FUNCTION_BLOCK Separator (* Basic Function Block Type *)
  (* Standard: 61499-2 *)
  (* Version 0.0, 2015-03-24, 4DIAC-IDE, 4DIAC-Consortium *)
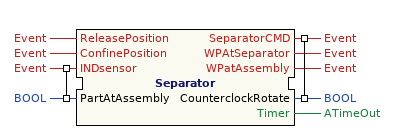
  EVENT_INPUT
    ReleasePosition;
    ConfinePosition;
    INDsensor WITH PartAtAssembly;
  END_EVENT
  EVENT_OUTPUT
    SeparatorCMD WITH CounterclockRotate;
    WPAtSeparator;
    WPatAssembly;
  END_EVENT
  VAR_INPUT
    PartAtAssembly : BOOL;
  END_VAR
  VAR_OUTPUT
    CounterclockRotate : BOOL;
  END_VAR
  PLUGS
    Timer : ATimeOut;
  END_PLUGS
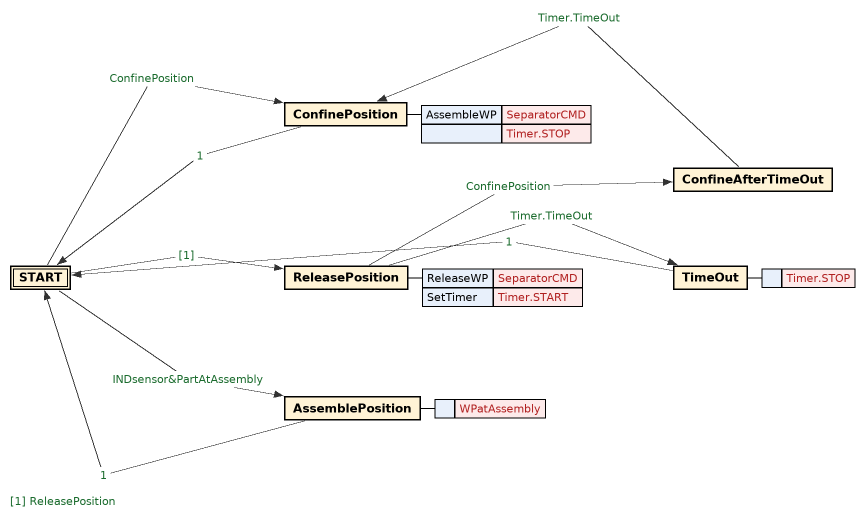
  EC_STATES
    START; (* Initial State *)
    ReleasePosition : ReleaseWP -> SeparatorCMD, SetTimer -> Timer.START;
    AssemblePosition : -> WPatAssembly;
    ConfinePosition : AssembleWP -> SeparatorCMD, -> Timer.STOP;
    TimeOut : -> Timer.STOP;
    ConfineAfterTimeOut;
  END_STATES
  EC_TRANSITIONS
    START TO ReleasePosition := ReleasePosition;
    ConfinePosition TO START := 1;
    AssemblePosition TO START := 1;
    TimeOut TO START := 1;
    ReleasePosition TO TimeOut := Timer.TimeOut;
    START TO AssemblePosition := INDsensor&PartAtAssembly;
    START TO ConfinePosition := ConfinePosition;
    ReleasePosition TO ConfineAfterTimeOut := ConfinePosition;
    ConfineAfterTimeOut TO ConfinePosition := Timer.TimeOut;
  END_TRANSITIONS
  ALGORITHM ReleaseWP IN ST:
CounterclockRotate := FALSE;
  END_ALGORITHM
  ALGORITHM AssembleWP IN ST:
CounterclockRotate := TRUE;
  END_ALGORITHM
  ALGORITHM SetTimer IN ST: (* new algorithm *)
Timer.DT := T#750ms;
  END_ALGORITHM
  SERVICE separator_interface/separator_implementation (* Basic Function Block Type *)
    SEQUENCE ReleasePosition_Timer
      separator_interface.ReleasePosition() -> separator_interface.SeparatorCMD(CounterclockRotate = false) -> separator_interface.Timer.START(Timer.DT = T#750ms);
      separator_interface.Timer.TimeOut() -> separator_interface.Timer.STOP();
    END_SEQUENCE
    SEQUENCE AssemblePosition
      separator_interface.INDsensor(PartAtAssembly = true) -> separator_interface.WPatAssembly();
    END_SEQUENCE
    SEQUENCE ConfinePosition
      separator_interface.ConfinePosition() -> separator_interface.SeparatorCMD(CounterclockRotate = true) -> separator_interface.Timer.STOP();
    END_SEQUENCE
    SEQUENCE ReleasePosition_Confine
      separator_interface.ReleasePosition() -> separator_interface.SeparatorCMD(CounterclockRotate = false) -> separator_interface.Timer.START(Timer.DT = T#750ms);
      separator_interface.ConfinePosition();
      separator_interface.Timer.TimeOut() -> separator_interface.SeparatorCMD(CounterclockRotate = true) -> separator_interface.Timer.STOP();
    END_SEQUENCE
  END_SERVICE
END_FUNCTION_BLOCK
